TYPE stSettings_Camera :
STRUCT
	aCameraMatrix : TcVnMatrix3x3_LREAL;
    aDistortionCoefficients : TcVnArray8_LREAL;
	UseParamFile : BOOL := TRUE;
	sFilePath: STRING;
END_STRUCT
END_TYPE

(* stored: Version 1.1.0.1, ProductVersion 3.1.4026.18
   DUT stSettings_Camera: Id {4aede540-508f-4dd9-96e9-57227feb46e2} *)
